PROGRAM MAIN
VAR
	timer : ULINT;
END_VAR

timer := timer + 2;

END_PROGRAM

(* stored: Version 1.1.0.1, ProductVersion 3.1.4024.12
   POU MAIN: Id {b051a9b6-3725-4d1f-b3dd-6053249d9316}, SpecialFunc None *)
